(* CODESYS project CtaVisSymbols_2.0.0.0.library
   DocFormat: reStructuredText
   DefaultNamespace: CtaVisSymbols
   Version: 2.0.0.0
   Placeholder: CtaVisSymbols
   Company: CTA
   Description: Symbol Library der CTA
   CompiledLibraryCompatibilityVersion: CODESYS V3.5 SP16 Patch 3
   LanguageModelAttribute: qualified-access-only
   Title: CtaVisSymbols
   Author: SIS

Project tree, tasks and I/O mapping:
  libraries: CmpBitmapPool, 3.5.17.0 (System); VisuSymbols, 4.5.0.0 (System)
  40 Visualizations/
  30 Program Organization Units/
  00000000-0000-0000-0000-000000000000|D:\CoDeSys\LibrariesV3\trunk\Intern\CAA\CAA Template\3.4.0.0 draft\Placeholder.xml
  00000000-0000-0000-0000-000000000000|D:\CoDeSys\LibrariesV3\trunk\Intern\CAA\CAA Template\3.2.0.3 draft\Prefix.pdf
  00000000-0000-0000-0000-000000000000|D:\CoDeSys\LibrariesV3\trunk\Intern\CAA\CAA Template\3.5.2.0 draft\Placeholder.xml
  20 Structs/
  50 Images/
    image pool ImagePool
  10 Documenation/
    global variables VersionHistory
    global variables readMe
  21 Interface/
  11 Library Parameter/
  12 Konstanten/
  60 Textlisten/
  13 Globale Variablen/
  5ce3da45-db07-42e7-a21c-a00fff4ed8f6|Icons\Account.svg
  5ce3da45-db07-42e7-a21c-a00fff4ed8f6|Icons\alert.svg
  5ce3da45-db07-42e7-a21c-a00fff4ed8f6|Icons\alert_solo_black.svg
  5ce3da45-db07-42e7-a21c-a00fff4ed8f6|Icons\arrow-down.svg
  5ce3da45-db07-42e7-a21c-a00fff4ed8f6|Icons\arrow-down_solo_black.svg
  5ce3da45-db07-42e7-a21c-a00fff4ed8f6|Icons\arrow-down_square.svg
  5ce3da45-db07-42e7-a21c-a00fff4ed8f6|Icons\arrow-left.svg
  5ce3da45-db07-42e7-a21c-a00fff4ed8f6|Icons\arrow-left_solo_black.svg
  5ce3da45-db07-42e7-a21c-a00fff4ed8f6|Icons\arrow-left_square.svg
  5ce3da45-db07-42e7-a21c-a00fff4ed8f6|Icons\arrow-right_solo_black.svg
  5ce3da45-db07-42e7-a21c-a00fff4ed8f6|Icons\arrow-right_square.svg
  5ce3da45-db07-42e7-a21c-a00fff4ed8f6|Icons\arrow-up.svg
  5ce3da45-db07-42e7-a21c-a00fff4ed8f6|Icons\build.svg
  5ce3da45-db07-42e7-a21c-a00fff4ed8f6|Icons\calendar-range.svg
  5ce3da45-db07-42e7-a21c-a00fff4ed8f6|Icons\chart-bell-curve.svg
  5ce3da45-db07-42e7-a21c-a00fff4ed8f6|Icons\check.svg
  5ce3da45-db07-42e7-a21c-a00fff4ed8f6|Icons\check_solo_black.svg
  5ce3da45-db07-42e7-a21c-a00fff4ed8f6|Icons\clock-outline.svg
  5ce3da45-db07-42e7-a21c-a00fff4ed8f6|Icons\close.svg
  5ce3da45-db07-42e7-a21c-a00fff4ed8f6|Icons\close_solo_black.svg
  5ce3da45-db07-42e7-a21c-a00fff4ed8f6|Icons\CtaError.svg
  5ce3da45-db07-42e7-a21c-a00fff4ed8f6|Icons\CtaInfo.svg
  5ce3da45-db07-42e7-a21c-a00fff4ed8f6|Icons\CtaWarning.svg
  5ce3da45-db07-42e7-a21c-a00fff4ed8f6|Icons\database_black.svg
  5ce3da45-db07-42e7-a21c-a00fff4ed8f6|Icons\delete.svg
  5ce3da45-db07-42e7-a21c-a00fff4ed8f6|Icons\delete_solo_black.svg
  5ce3da45-db07-42e7-a21c-a00fff4ed8f6|Icons\dip-switch.svg
  5ce3da45-db07-42e7-a21c-a00fff4ed8f6|Icons\engine.svg
  5ce3da45-db07-42e7-a21c-a00fff4ed8f6|Icons\eye.svg
  5ce3da45-db07-42e7-a21c-a00fff4ed8f6|Icons\front_hand_Black.svg
  5ce3da45-db07-42e7-a21c-a00fff4ed8f6|Icons\front_hand_Yellow.svg
  5ce3da45-db07-42e7-a21c-a00fff4ed8f6|Icons\front_hand_Yellow_Off.svg
  5ce3da45-db07-42e7-a21c-a00fff4ed8f6|Icons\functions_black_24dp.svg
  5ce3da45-db07-42e7-a21c-a00fff4ed8f6|Icons\gear.svg
  5ce3da45-db07-42e7-a21c-a00fff4ed8f6|Icons\help.svg
  5ce3da45-db07-42e7-a21c-a00fff4ed8f6|Icons\home.svg
  5ce3da45-db07-42e7-a21c-a00fff4ed8f6|Icons\home_solo_black.svg
  5ce3da45-db07-42e7-a21c-a00fff4ed8f6|Icons\information-variant.svg
  5ce3da45-db07-42e7-a21c-a00fff4ed8f6|Icons\lan.svg
  5ce3da45-db07-42e7-a21c-a00fff4ed8f6|Icons\lightning-bolt-circle.svg
  5ce3da45-db07-42e7-a21c-a00fff4ed8f6|Icons\menu.svg
  5ce3da45-db07-42e7-a21c-a00fff4ed8f6|Icons\message.svg
  5ce3da45-db07-42e7-a21c-a00fff4ed8f6|Icons\message-alert-variant red.svg
  5ce3da45-db07-42e7-a21c-a00fff4ed8f6|Icons\message-alert-variant.svg
  5ce3da45-db07-42e7-a21c-a00fff4ed8f6|Icons\minus.svg
  5ce3da45-db07-42e7-a21c-a00fff4ed8f6|Icons\minus_solo_black.svg
  5ce3da45-db07-42e7-a21c-a00fff4ed8f6|Icons\plus.svg
  5ce3da45-db07-42e7-a21c-a00fff4ed8f6|Icons\plus_solo_black.svg
  5ce3da45-db07-42e7-a21c-a00fff4ed8f6|Icons\power.svg
  5ce3da45-db07-42e7-a21c-a00fff4ed8f6|Icons\power_solo_black.svg
  5ce3da45-db07-42e7-a21c-a00fff4ed8f6|Icons\refresh.svg
  5ce3da45-db07-42e7-a21c-a00fff4ed8f6|Icons\refresh_solo_black.svg
  5ce3da45-db07-42e7-a21c-a00fff4ed8f6|Icons\sd_card_black_24dp.svg
  5ce3da45-db07-42e7-a21c-a00fff4ed8f6|Icons\SearchFilter.svg
  5ce3da45-db07-42e7-a21c-a00fff4ed8f6|Icons\settings.svg
  5ce3da45-db07-42e7-a21c-a00fff4ed8f6|Icons\signal-celular-alt.svg
  5ce3da45-db07-42e7-a21c-a00fff4ed8f6|Icons\sine-wave.svg
  5ce3da45-db07-42e7-a21c-a00fff4ed8f6|Icons\toggle-switch.svg
  5ce3da45-db07-42e7-a21c-a00fff4ed8f6|Icons\toggle-switch-off.svg
  5ce3da45-db07-42e7-a21c-a00fff4ed8f6|Icons\Modbus_Organization_Logo.svg
  5ce3da45-db07-42e7-a21c-a00fff4ed8f6|Icons\CheckboxChecked_blue.svg
  5ce3da45-db07-42e7-a21c-a00fff4ed8f6|Icons\CheckboxUnchecked_withe.svg
  5ce3da45-db07-42e7-a21c-a00fff4ed8f6|Icons\lock_closed_black.svg
  5ce3da45-db07-42e7-a21c-a00fff4ed8f6|Icons\lock_open_black.svg
  5ce3da45-db07-42e7-a21c-a00fff4ed8f6|Icons\check_green.svg
  5ce3da45-db07-42e7-a21c-a00fff4ed8f6|Icons\close_red.svg
  5ce3da45-db07-42e7-a21c-a00fff4ed8f6|Icons\Sensor_Black.svg
  5ce3da45-db07-42e7-a21c-a00fff4ed8f6|Icons\filter_black.svg
  5ce3da45-db07-42e7-a21c-a00fff4ed8f6|Icons\notification_black.svg
  5ce3da45-db07-42e7-a21c-a00fff4ed8f6|Icons\CtaLogo.png
  5ce3da45-db07-42e7-a21c-a00fff4ed8f6|Icons\Edit_Stift.svg
  5ce3da45-db07-42e7-a21c-a00fff4ed8f6|Icons\Grafana_Logo.svg
  5ce3da45-db07-42e7-a21c-a00fff4ed8f6|Icons\InfluxDb_Logo.svg
  5ce3da45-db07-42e7-a21c-a00fff4ed8f6|Icons\hourglass_top.svg
  5ce3da45-db07-42e7-a21c-a00fff4ed8f6|Icons\Settings+.svg
  5ce3da45-db07-42e7-a21c-a00fff4ed8f6|Icons\Hourglass.gif
  5ce3da45-db07-42e7-a21c-a00fff4ed8f6|Icons\HandTapAwake.svg
  5ce3da45-db07-42e7-a21c-a00fff4ed8f6|Icons\gear_white.svg
  5ce3da45-db07-42e7-a21c-a00fff4ed8f6|S:\_Temporär_SIS\CtaCodesysLibrary\01_Library\CtaVisSymbols\Icons\SettingsSmall.svg
  5ce3da45-db07-42e7-a21c-a00fff4ed8f6|S:\_Temporär_SIS\CtaCodesysLibrary\01_Library\CtaVisSymbols\Icons\FileDescription.svg
  5ce3da45-db07-42e7-a21c-a00fff4ed8f6|S:\_Temporär_SIS\CtaCodesysLibrary\01_Library\CtaVisSymbols\Icons\Modbus_Organization_Logo_Short.svg
  5ce3da45-db07-42e7-a21c-a00fff4ed8f6|S:\_Temporär_SIS\CtaCodesysLibrary\01_Library\CtaVisSymbols\Icons\Chart.svg
  5ce3da45-db07-42e7-a21c-a00fff4ed8f6|\\cta.local\mue\Daten\200_Klima_Kälte\200_300_KK_CTA_Exklusiv_Elektro\01_Elektro\03_Software\00_CtaCodesysLibrary\01_Library\01 Source Code\CtaVisSymbols\Icons\ac_unit_40dp_ffffff_fill0_wght400_grad0_opsz40.svg
  5ce3da45-db07-42e7-a21c-a00fff4ed8f6|P:\200_Klima_Kälte\200_300_KK_CTA_Exklusiv_Elektro\01_Elektro\03_Software\00_CtaCodesysLibrary\01_Library\CtaVisSymbols\Icons\Account.svg
  5ce3da45-db07-42e7-a21c-a00fff4ed8f6|P:\200_Klima_Kälte\200_300_KK_CTA_Exklusiv_Elektro\01_Elektro\03_Software\00_CtaCodesysLibrary\01_Library\CtaVisSymbols\Icons\alert.svg
  5ce3da45-db07-42e7-a21c-a00fff4ed8f6|P:\200_Klima_Kälte\200_300_KK_CTA_Exklusiv_Elektro\01_Elektro\03_Software\00_CtaCodesysLibrary\01_Library\CtaVisSymbols\Icons\alert_solo_black.svg
  5ce3da45-db07-42e7-a21c-a00fff4ed8f6|P:\200_Klima_Kälte\200_300_KK_CTA_Exklusiv_Elektro\01_Elektro\03_Software\00_CtaCodesysLibrary\01_Library\CtaVisSymbols\Icons\arrow-down.svg
  5ce3da45-db07-42e7-a21c-a00fff4ed8f6|P:\200_Klima_Kälte\200_300_KK_CTA_Exklusiv_Elektro\01_Elektro\03_Software\00_CtaCodesysLibrary\01_Library\CtaVisSymbols\Icons\arrow-down_solo_black.svg
  5ce3da45-db07-42e7-a21c-a00fff4ed8f6|P:\200_Klima_Kälte\200_300_KK_CTA_Exklusiv_Elektro\01_Elektro\03_Software\00_CtaCodesysLibrary\01_Library\CtaVisSymbols\Icons\arrow-down_square.svg
  5ce3da45-db07-42e7-a21c-a00fff4ed8f6|P:\200_Klima_Kälte\200_300_KK_CTA_Exklusiv_Elektro\01_Elektro\03_Software\00_CtaCodesysLibrary\01_Library\CtaVisSymbols\Icons\arrow-left.svg
  5ce3da45-db07-42e7-a21c-a00fff4ed8f6|P:\200_Klima_Kälte\200_300_KK_CTA_Exklusiv_Elektro\01_Elektro\03_Software\00_CtaCodesysLibrary\01_Library\CtaVisSymbols\Icons\arrow-left_solo_black.svg
  5ce3da45-db07-42e7-a21c-a00fff4ed8f6|P:\200_Klima_Kälte\200_300_KK_CTA_Exklusiv_Elektro\01_Elektro\03_Software\00_CtaCodesysLibrary\01_Library\CtaVisSymbols\Icons\arrow-left_square.svg
  5ce3da45-db07-42e7-a21c-a00fff4ed8f6|P:\200_Klima_Kälte\200_300_KK_CTA_Exklusiv_Elektro\01_Elektro\03_Software\00_CtaCodesysLibrary\01_Library\CtaVisSymbols\Icons\arrow-right_solo_black.svg
  5ce3da45-db07-42e7-a21c-a00fff4ed8f6|P:\200_Klima_Kälte\200_300_KK_CTA_Exklusiv_Elektro\01_Elektro\03_Software\00_CtaCodesysLibrary\01_Library\CtaVisSymbols\Icons\arrow-right_square.svg
  5ce3da45-db07-42e7-a21c-a00fff4ed8f6|P:\200_Klima_Kälte\200_300_KK_CTA_Exklusiv_Elektro\01_Elektro\03_Software\00_CtaCodesysLibrary\01_Library\CtaVisSymbols\Icons\arrow-up.svg
  5ce3da45-db07-42e7-a21c-a00fff4ed8f6|P:\200_Klima_Kälte\200_300_KK_CTA_Exklusiv_Elektro\01_Elektro\03_Software\00_CtaCodesysLibrary\01_Library\CtaVisSymbols\Icons\build.svg
  5ce3da45-db07-42e7-a21c-a00fff4ed8f6|P:\200_Klima_Kälte\200_300_KK_CTA_Exklusiv_Elektro\01_Elektro\03_Software\00_CtaCodesysLibrary\01_Library\CtaVisSymbols\Icons\calendar-range.svg
  5ce3da45-db07-42e7-a21c-a00fff4ed8f6|P:\200_Klima_Kälte\200_300_KK_CTA_Exklusiv_Elektro\01_Elektro\03_Software\00_CtaCodesysLibrary\01_Library\CtaVisSymbols\Icons\Chart.svg
  5ce3da45-db07-42e7-a21c-a00fff4ed8f6|P:\200_Klima_Kälte\200_300_KK_CTA_Exklusiv_Elektro\01_Elektro\03_Software\00_CtaCodesysLibrary\01_Library\CtaVisSymbols\Icons\chart-bell-curve.svg
  5ce3da45-db07-42e7-a21c-a00fff4ed8f6|P:\200_Klima_Kälte\200_300_KK_CTA_Exklusiv_Elektro\01_Elektro\03_Software\00_CtaCodesysLibrary\01_Library\CtaVisSymbols\Icons\ChartLine.svg
  5ce3da45-db07-42e7-a21c-a00fff4ed8f6|P:\200_Klima_Kälte\200_300_KK_CTA_Exklusiv_Elektro\01_Elektro\03_Software\00_CtaCodesysLibrary\01_Library\CtaVisSymbols\Icons\chat_bubble_40dp_ffffff_fill0_wght400_grad0_opsz40.svg
  5ce3da45-db07-42e7-a21c-a00fff4ed8f6|P:\200_Klima_Kälte\200_300_KK_CTA_Exklusiv_Elektro\01_Elektro\03_Software\00_CtaCodesysLibrary\01_Library\CtaVisSymbols\Icons\check.svg
  5ce3da45-db07-42e7-a21c-a00fff4ed8f6|P:\200_Klima_Kälte\200_300_KK_CTA_Exklusiv_Elektro\01_Elektro\03_Software\00_CtaCodesysLibrary\01_Library\CtaVisSymbols\Icons\check_green.svg
  5ce3da45-db07-42e7-a21c-a00fff4ed8f6|P:\200_Klima_Kälte\200_300_KK_CTA_Exklusiv_Elektro\01_Elektro\03_Software\00_CtaCodesysLibrary\01_Library\CtaVisSymbols\Icons\check_solo_black.svg
  5ce3da45-db07-42e7-a21c-a00fff4ed8f6|P:\200_Klima_Kälte\200_300_KK_CTA_Exklusiv_Elektro\01_Elektro\03_Software\00_CtaCodesysLibrary\01_Library\CtaVisSymbols\Icons\checkboxchecked.svg
  5ce3da45-db07-42e7-a21c-a00fff4ed8f6|P:\200_Klima_Kälte\200_300_KK_CTA_Exklusiv_Elektro\01_Elektro\03_Software\00_CtaCodesysLibrary\01_Library\CtaVisSymbols\Icons\CheckboxChecked_blue.svg
  5ce3da45-db07-42e7-a21c-a00fff4ed8f6|P:\200_Klima_Kälte\200_300_KK_CTA_Exklusiv_Elektro\01_Elektro\03_Software\00_CtaCodesysLibrary\01_Library\CtaVisSymbols\Icons\checkboxchecked_def.svg
  5ce3da45-db07-42e7-a21c-a00fff4ed8f6|P:\200_Klima_Kälte\200_300_KK_CTA_Exklusiv_Elektro\01_Elektro\03_Software\00_CtaCodesysLibrary\01_Library\CtaVisSymbols\Icons\checkboxunchecked.svg
  5ce3da45-db07-42e7-a21c-a00fff4ed8f6|P:\200_Klima_Kälte\200_300_KK_CTA_Exklusiv_Elektro\01_Elektro\03_Software\00_CtaCodesysLibrary\01_Library\CtaVisSymbols\Icons\checkboxunchecked_def.svg
  5ce3da45-db07-42e7-a21c-a00fff4ed8f6|P:\200_Klima_Kälte\200_300_KK_CTA_Exklusiv_Elektro\01_Elektro\03_Software\00_CtaCodesysLibrary\01_Library\CtaVisSymbols\Icons\CheckboxUnchecked_withe.svg
  5ce3da45-db07-42e7-a21c-a00fff4ed8f6|P:\200_Klima_Kälte\200_300_KK_CTA_Exklusiv_Elektro\01_Elektro\03_Software\00_CtaCodesysLibrary\01_Library\CtaVisSymbols\Icons\clock-outline.svg
  5ce3da45-db07-42e7-a21c-a00fff4ed8f6|P:\200_Klima_Kälte\200_300_KK_CTA_Exklusiv_Elektro\01_Elektro\03_Software\00_CtaCodesysLibrary\01_Library\CtaVisSymbols\Icons\close.svg
  5ce3da45-db07-42e7-a21c-a00fff4ed8f6|P:\200_Klima_Kälte\200_300_KK_CTA_Exklusiv_Elektro\01_Elektro\03_Software\00_CtaCodesysLibrary\01_Library\CtaVisSymbols\Icons\close_red.svg
  5ce3da45-db07-42e7-a21c-a00fff4ed8f6|P:\200_Klima_Kälte\200_300_KK_CTA_Exklusiv_Elektro\01_Elektro\03_Software\00_CtaCodesysLibrary\01_Library\CtaVisSymbols\Icons\close_solo_black.svg
  5ce3da45-db07-42e7-a21c-a00fff4ed8f6|P:\200_Klima_Kälte\200_300_KK_CTA_Exklusiv_Elektro\01_Elektro\03_Software\00_CtaCodesysLibrary\01_Library\CtaVisSymbols\Icons\cloud_24dp_ffffff_fill0_wght400_grad0_opsz24.svg
  5ce3da45-db07-42e7-a21c-a00fff4ed8f6|P:\200_Klima_Kälte\200_300_KK_CTA_Exklusiv_Elektro\01_Elektro\03_Software\00_CtaCodesysLibrary\01_Library\CtaVisSymbols\Icons\cloudy_snowing_24dp_ffffff_fill0_wght400_grad0_opsz24.svg
  5ce3da45-db07-42e7-a21c-a00fff4ed8f6|P:\200_Klima_Kälte\200_300_KK_CTA_Exklusiv_Elektro\01_Elektro\03_Software\00_CtaCodesysLibrary\01_Library\CtaVisSymbols\Icons\CtaError.svg
  5ce3da45-db07-42e7-a21c-a00fff4ed8f6|P:\200_Klima_Kälte\200_300_KK_CTA_Exklusiv_Elektro\01_Elektro\03_Software\00_CtaCodesysLibrary\01_Library\CtaVisSymbols\Icons\CtaInfo.svg
  5ce3da45-db07-42e7-a21c-a00fff4ed8f6|P:\200_Klima_Kälte\200_300_KK_CTA_Exklusiv_Elektro\01_Elektro\03_Software\00_CtaCodesysLibrary\01_Library\CtaVisSymbols\Icons\CtaLogo.png
  5ce3da45-db07-42e7-a21c-a00fff4ed8f6|P:\200_Klima_Kälte\200_300_KK_CTA_Exklusiv_Elektro\01_Elektro\03_Software\00_CtaCodesysLibrary\01_Library\CtaVisSymbols\Icons\CtaWarning.svg
  5ce3da45-db07-42e7-a21c-a00fff4ed8f6|P:\200_Klima_Kälte\200_300_KK_CTA_Exklusiv_Elektro\01_Elektro\03_Software\00_CtaCodesysLibrary\01_Library\CtaVisSymbols\Icons\database_black.svg
  5ce3da45-db07-42e7-a21c-a00fff4ed8f6|P:\200_Klima_Kälte\200_300_KK_CTA_Exklusiv_Elektro\01_Elektro\03_Software\00_CtaCodesysLibrary\01_Library\CtaVisSymbols\Icons\delete.svg
  5ce3da45-db07-42e7-a21c-a00fff4ed8f6|P:\200_Klima_Kälte\200_300_KK_CTA_Exklusiv_Elektro\01_Elektro\03_Software\00_CtaCodesysLibrary\01_Library\CtaVisSymbols\Icons\delete_solo_black.svg
  5ce3da45-db07-42e7-a21c-a00fff4ed8f6|P:\200_Klima_Kälte\200_300_KK_CTA_Exklusiv_Elektro\01_Elektro\03_Software\00_CtaCodesysLibrary\01_Library\CtaVisSymbols\Icons\dictionary_40dp_ffffff_fill0_wght400_grad0_opsz40.svg
  5ce3da45-db07-42e7-a21c-a00fff4ed8f6|P:\200_Klima_Kälte\200_300_KK_CTA_Exklusiv_Elektro\01_Elektro\03_Software\00_CtaCodesysLibrary\01_Library\CtaVisSymbols\Icons\dip-switch.svg
  5ce3da45-db07-42e7-a21c-a00fff4ed8f6|P:\200_Klima_Kälte\200_300_KK_CTA_Exklusiv_Elektro\01_Elektro\03_Software\00_CtaCodesysLibrary\01_Library\CtaVisSymbols\Icons\Edit_Stift.svg
  5ce3da45-db07-42e7-a21c-a00fff4ed8f6|P:\200_Klima_Kälte\200_300_KK_CTA_Exklusiv_Elektro\01_Elektro\03_Software\00_CtaCodesysLibrary\01_Library\CtaVisSymbols\Icons\electric_bolt_24dp_000000_FILL0_wght400_GRAD0_opsz24.svg
  5ce3da45-db07-42e7-a21c-a00fff4ed8f6|P:\200_Klima_Kälte\200_300_KK_CTA_Exklusiv_Elektro\01_Elektro\03_Software\00_CtaCodesysLibrary\01_Library\CtaVisSymbols\Icons\engine.svg
  5ce3da45-db07-42e7-a21c-a00fff4ed8f6|P:\200_Klima_Kälte\200_300_KK_CTA_Exklusiv_Elektro\01_Elektro\03_Software\00_CtaCodesysLibrary\01_Library\CtaVisSymbols\Icons\engineering_40dp_ffffff_fill0_wght400_grad0_opsz40.svg
  5ce3da45-db07-42e7-a21c-a00fff4ed8f6|P:\200_Klima_Kälte\200_300_KK_CTA_Exklusiv_Elektro\01_Elektro\03_Software\00_CtaCodesysLibrary\01_Library\CtaVisSymbols\Icons\eye.svg
  5ce3da45-db07-42e7-a21c-a00fff4ed8f6|P:\200_Klima_Kälte\200_300_KK_CTA_Exklusiv_Elektro\01_Elektro\03_Software\00_CtaCodesysLibrary\01_Library\CtaVisSymbols\Icons\FileDescription.svg
  5ce3da45-db07-42e7-a21c-a00fff4ed8f6|P:\200_Klima_Kälte\200_300_KK_CTA_Exklusiv_Elektro\01_Elektro\03_Software\00_CtaCodesysLibrary\01_Library\CtaVisSymbols\Icons\filter_black.svg
  5ce3da45-db07-42e7-a21c-a00fff4ed8f6|P:\200_Klima_Kälte\200_300_KK_CTA_Exklusiv_Elektro\01_Elektro\03_Software\00_CtaCodesysLibrary\01_Library\CtaVisSymbols\Icons\foggy_24dp_ffffff_fill0_wght400_grad0_opsz24.svg
  5ce3da45-db07-42e7-a21c-a00fff4ed8f6|P:\200_Klima_Kälte\200_300_KK_CTA_Exklusiv_Elektro\01_Elektro\03_Software\00_CtaCodesysLibrary\01_Library\CtaVisSymbols\Icons\folder.svg
  5ce3da45-db07-42e7-a21c-a00fff4ed8f6|P:\200_Klima_Kälte\200_300_KK_CTA_Exklusiv_Elektro\01_Elektro\03_Software\00_CtaCodesysLibrary\01_Library\CtaVisSymbols\Icons\front_hand_Black.svg
  5ce3da45-db07-42e7-a21c-a00fff4ed8f6|P:\200_Klima_Kälte\200_300_KK_CTA_Exklusiv_Elektro\01_Elektro\03_Software\00_CtaCodesysLibrary\01_Library\CtaVisSymbols\Icons\front_hand_Yellow.svg
  5ce3da45-db07-42e7-a21c-a00fff4ed8f6|P:\200_Klima_Kälte\200_300_KK_CTA_Exklusiv_Elektro\01_Elektro\03_Software\00_CtaCodesysLibrary\01_Library\CtaVisSymbols\Icons\front_hand_Yellow_Off.svg
  5ce3da45-db07-42e7-a21c-a00fff4ed8f6|P:\200_Klima_Kälte\200_300_KK_CTA_Exklusiv_Elektro\01_Elektro\03_Software\00_CtaCodesysLibrary\01_Library\CtaVisSymbols\Icons\functions_black_24dp.svg
  5ce3da45-db07-42e7-a21c-a00fff4ed8f6|P:\200_Klima_Kälte\200_300_KK_CTA_Exklusiv_Elektro\01_Elektro\03_Software\00_CtaCodesysLibrary\01_Library\CtaVisSymbols\Icons\gear.svg
  5ce3da45-db07-42e7-a21c-a00fff4ed8f6|P:\200_Klima_Kälte\200_300_KK_CTA_Exklusiv_Elektro\01_Elektro\03_Software\00_CtaCodesysLibrary\01_Library\CtaVisSymbols\Icons\gear_white.svg
  5ce3da45-db07-42e7-a21c-a00fff4ed8f6|P:\200_Klima_Kälte\200_300_KK_CTA_Exklusiv_Elektro\01_Elektro\03_Software\00_CtaCodesysLibrary\01_Library\CtaVisSymbols\Icons\Grafana_Logo.svg
  5ce3da45-db07-42e7-a21c-a00fff4ed8f6|P:\200_Klima_Kälte\200_300_KK_CTA_Exklusiv_Elektro\01_Elektro\03_Software\00_CtaCodesysLibrary\01_Library\CtaVisSymbols\Icons\HandTapAwake.svg
  5ce3da45-db07-42e7-a21c-a00fff4ed8f6|P:\200_Klima_Kälte\200_300_KK_CTA_Exklusiv_Elektro\01_Elektro\03_Software\00_CtaCodesysLibrary\01_Library\CtaVisSymbols\Icons\help.svg
  5ce3da45-db07-42e7-a21c-a00fff4ed8f6|P:\200_Klima_Kälte\200_300_KK_CTA_Exklusiv_Elektro\01_Elektro\03_Software\00_CtaCodesysLibrary\01_Library\CtaVisSymbols\Icons\home.svg
  5ce3da45-db07-42e7-a21c-a00fff4ed8f6|P:\200_Klima_Kälte\200_300_KK_CTA_Exklusiv_Elektro\01_Elektro\03_Software\00_CtaCodesysLibrary\01_Library\CtaVisSymbols\Icons\home_40dp_ffffff_fill0_wght400_grad0_opsz40.svg
  5ce3da45-db07-42e7-a21c-a00fff4ed8f6|P:\200_Klima_Kälte\200_300_KK_CTA_Exklusiv_Elektro\01_Elektro\03_Software\00_CtaCodesysLibrary\01_Library\CtaVisSymbols\Icons\home_solo_black.svg
  5ce3da45-db07-42e7-a21c-a00fff4ed8f6|P:\200_Klima_Kälte\200_300_KK_CTA_Exklusiv_Elektro\01_Elektro\03_Software\00_CtaCodesysLibrary\01_Library\CtaVisSymbols\Icons\Hourglass.gif
  5ce3da45-db07-42e7-a21c-a00fff4ed8f6|P:\200_Klima_Kälte\200_300_KK_CTA_Exklusiv_Elektro\01_Elektro\03_Software\00_CtaCodesysLibrary\01_Library\CtaVisSymbols\Icons\hourglass_top.svg
  5ce3da45-db07-42e7-a21c-a00fff4ed8f6|P:\200_Klima_Kälte\200_300_KK_CTA_Exklusiv_Elektro\01_Elektro\03_Software\00_CtaCodesysLibrary\01_Library\CtaVisSymbols\Icons\hub_20dp_ffffff_fill0_wght400_grad0_opsz20.svg
  5ce3da45-db07-42e7-a21c-a00fff4ed8f6|P:\200_Klima_Kälte\200_300_KK_CTA_Exklusiv_Elektro\01_Elektro\03_Software\00_CtaCodesysLibrary\01_Library\CtaVisSymbols\Icons\InfluxDb_Logo.svg
  5ce3da45-db07-42e7-a21c-a00fff4ed8f6|P:\200_Klima_Kälte\200_300_KK_CTA_Exklusiv_Elektro\01_Elektro\03_Software\00_CtaCodesysLibrary\01_Library\CtaVisSymbols\Icons\information-variant.svg
  5ce3da45-db07-42e7-a21c-a00fff4ed8f6|P:\200_Klima_Kälte\200_300_KK_CTA_Exklusiv_Elektro\01_Elektro\03_Software\00_CtaCodesysLibrary\01_Library\CtaVisSymbols\Icons\instant_mix_40dp_ffffff_fill0_wght400_grad0_opsz40.svg
  5ce3da45-db07-42e7-a21c-a00fff4ed8f6|P:\200_Klima_Kälte\200_300_KK_CTA_Exklusiv_Elektro\01_Elektro\03_Software\00_CtaCodesysLibrary\01_Library\CtaVisSymbols\Icons\lan.svg
  5ce3da45-db07-42e7-a21c-a00fff4ed8f6|P:\200_Klima_Kälte\200_300_KK_CTA_Exklusiv_Elektro\01_Elektro\03_Software\00_CtaCodesysLibrary\01_Library\CtaVisSymbols\Icons\lan_40dp_ffffff_fill0_wght400_grad0_opsz40.svg
  5ce3da45-db07-42e7-a21c-a00fff4ed8f6|P:\200_Klima_Kälte\200_300_KK_CTA_Exklusiv_Elektro\01_Elektro\03_Software\00_CtaCodesysLibrary\01_Library\CtaVisSymbols\Icons\language_50dp_ffffff_fill0_wght400_grad0_opsz48.svg
  5ce3da45-db07-42e7-a21c-a00fff4ed8f6|P:\200_Klima_Kälte\200_300_KK_CTA_Exklusiv_Elektro\01_Elektro\03_Software\00_CtaCodesysLibrary\01_Library\CtaVisSymbols\Icons\lightning-bolt-circle.svg
  5ce3da45-db07-42e7-a21c-a00fff4ed8f6|P:\200_Klima_Kälte\200_300_KK_CTA_Exklusiv_Elektro\01_Elektro\03_Software\00_CtaCodesysLibrary\01_Library\CtaVisSymbols\Icons\link_24dp_5f6368_fill0_wght400_grad0_opsz24.svg
  5ce3da45-db07-42e7-a21c-a00fff4ed8f6|P:\200_Klima_Kälte\200_300_KK_CTA_Exklusiv_Elektro\01_Elektro\03_Software\00_CtaCodesysLibrary\01_Library\CtaVisSymbols\Icons\link_off_24dp_5f6368_fill0_wght400_grad0_opsz24.svg
  5ce3da45-db07-42e7-a21c-a00fff4ed8f6|P:\200_Klima_Kälte\200_300_KK_CTA_Exklusiv_Elektro\01_Elektro\03_Software\00_CtaCodesysLibrary\01_Library\CtaVisSymbols\Icons\lock_closed_black.svg
  5ce3da45-db07-42e7-a21c-a00fff4ed8f6|P:\200_Klima_Kälte\200_300_KK_CTA_Exklusiv_Elektro\01_Elektro\03_Software\00_CtaCodesysLibrary\01_Library\CtaVisSymbols\Icons\lock_open_black.svg
  5ce3da45-db07-42e7-a21c-a00fff4ed8f6|P:\200_Klima_Kälte\200_300_KK_CTA_Exklusiv_Elektro\01_Elektro\03_Software\00_CtaCodesysLibrary\01_Library\CtaVisSymbols\Icons\lockicon.svg
  5ce3da45-db07-42e7-a21c-a00fff4ed8f6|P:\200_Klima_Kälte\200_300_KK_CTA_Exklusiv_Elektro\01_Elektro\03_Software\00_CtaCodesysLibrary\01_Library\CtaVisSymbols\Icons\logout_50dp_ffffff_fill0_wght400_grad0_opsz48.svg
  5ce3da45-db07-42e7-a21c-a00fff4ed8f6|P:\200_Klima_Kälte\200_300_KK_CTA_Exklusiv_Elektro\01_Elektro\03_Software\00_CtaCodesysLibrary\01_Library\CtaVisSymbols\Icons\memory_20dp_ffffff_fill0_wght400_grad0_opsz20.svg
  5ce3da45-db07-42e7-a21c-a00fff4ed8f6|P:\200_Klima_Kälte\200_300_KK_CTA_Exklusiv_Elektro\01_Elektro\03_Software\00_CtaCodesysLibrary\01_Library\CtaVisSymbols\Icons\menu.svg
  5ce3da45-db07-42e7-a21c-a00fff4ed8f6|P:\200_Klima_Kälte\200_300_KK_CTA_Exklusiv_Elektro\01_Elektro\03_Software\00_CtaCodesysLibrary\01_Library\CtaVisSymbols\Icons\menu_50dp_ffffff_fill0_wght400_grad0_opsz48.svg
  5ce3da45-db07-42e7-a21c-a00fff4ed8f6|P:\200_Klima_Kälte\200_300_KK_CTA_Exklusiv_Elektro\01_Elektro\03_Software\00_CtaCodesysLibrary\01_Library\CtaVisSymbols\Icons\menu_open_50dp_ffffff_fill0_wght400_grad0_opsz48.svg
  5ce3da45-db07-42e7-a21c-a00fff4ed8f6|P:\200_Klima_Kälte\200_300_KK_CTA_Exklusiv_Elektro\01_Elektro\03_Software\00_CtaCodesysLibrary\01_Library\CtaVisSymbols\Icons\message.svg
  5ce3da45-db07-42e7-a21c-a00fff4ed8f6|P:\200_Klima_Kälte\200_300_KK_CTA_Exklusiv_Elektro\01_Elektro\03_Software\00_CtaCodesysLibrary\01_Library\CtaVisSymbols\Icons\message-alert-variant red.svg
  5ce3da45-db07-42e7-a21c-a00fff4ed8f6|P:\200_Klima_Kälte\200_300_KK_CTA_Exklusiv_Elektro\01_Elektro\03_Software\00_CtaCodesysLibrary\01_Library\CtaVisSymbols\Icons\message-alert-variant.svg
  5ce3da45-db07-42e7-a21c-a00fff4ed8f6|P:\200_Klima_Kälte\200_300_KK_CTA_Exklusiv_Elektro\01_Elektro\03_Software\00_CtaCodesysLibrary\01_Library\CtaVisSymbols\Icons\minus.svg
  5ce3da45-db07-42e7-a21c-a00fff4ed8f6|P:\200_Klima_Kälte\200_300_KK_CTA_Exklusiv_Elektro\01_Elektro\03_Software\00_CtaCodesysLibrary\01_Library\CtaVisSymbols\Icons\minus_solo_black.svg
  5ce3da45-db07-42e7-a21c-a00fff4ed8f6|P:\200_Klima_Kälte\200_300_KK_CTA_Exklusiv_Elektro\01_Elektro\03_Software\00_CtaCodesysLibrary\01_Library\CtaVisSymbols\Icons\Modbus_Organization_Logo.svg
  5ce3da45-db07-42e7-a21c-a00fff4ed8f6|P:\200_Klima_Kälte\200_300_KK_CTA_Exklusiv_Elektro\01_Elektro\03_Software\00_CtaCodesysLibrary\01_Library\CtaVisSymbols\Icons\Modbus_Organization_Logo_Short.svg
  5ce3da45-db07-42e7-a21c-a00fff4ed8f6|P:\200_Klima_Kälte\200_300_KK_CTA_Exklusiv_Elektro\01_Elektro\03_Software\00_CtaCodesysLibrary\01_Library\CtaVisSymbols\Icons\mode_cool_24dp_ffffff_fill0_wght400_grad0_opsz24.svg
  5ce3da45-db07-42e7-a21c-a00fff4ed8f6|P:\200_Klima_Kälte\200_300_KK_CTA_Exklusiv_Elektro\01_Elektro\03_Software\00_CtaCodesysLibrary\01_Library\CtaVisSymbols\Icons\monitoring_40dp_ffffff_fill0_wght400_grad0_opsz40.svg
  5ce3da45-db07-42e7-a21c-a00fff4ed8f6|P:\200_Klima_Kälte\200_300_KK_CTA_Exklusiv_Elektro\01_Elektro\03_Software\00_CtaCodesysLibrary\01_Library\CtaVisSymbols\Icons\notification_black.svg
  5ce3da45-db07-42e7-a21c-a00fff4ed8f6|P:\200_Klima_Kälte\200_300_KK_CTA_Exklusiv_Elektro\01_Elektro\03_Software\00_CtaCodesysLibrary\01_Library\CtaVisSymbols\Icons\partly_cloudy_day_24dp_ffffff_fill0_wght400_grad0_opsz24.svg
  5ce3da45-db07-42e7-a21c-a00fff4ed8f6|P:\200_Klima_Kälte\200_300_KK_CTA_Exklusiv_Elektro\01_Elektro\03_Software\00_CtaCodesysLibrary\01_Library\CtaVisSymbols\Icons\person_50dp_ffffff_fill0_wght400_grad0_opsz48.svg
  5ce3da45-db07-42e7-a21c-a00fff4ed8f6|P:\200_Klima_Kälte\200_300_KK_CTA_Exklusiv_Elektro\01_Elektro\03_Software\00_CtaCodesysLibrary\01_Library\CtaVisSymbols\Icons\plus.svg
  5ce3da45-db07-42e7-a21c-a00fff4ed8f6|P:\200_Klima_Kälte\200_300_KK_CTA_Exklusiv_Elektro\01_Elektro\03_Software\00_CtaCodesysLibrary\01_Library\CtaVisSymbols\Icons\plus_solo_black.svg
  5ce3da45-db07-42e7-a21c-a00fff4ed8f6|P:\200_Klima_Kälte\200_300_KK_CTA_Exklusiv_Elektro\01_Elektro\03_Software\00_CtaCodesysLibrary\01_Library\CtaVisSymbols\Icons\power.svg
  5ce3da45-db07-42e7-a21c-a00fff4ed8f6|P:\200_Klima_Kälte\200_300_KK_CTA_Exklusiv_Elektro\01_Elektro\03_Software\00_CtaCodesysLibrary\01_Library\CtaVisSymbols\Icons\power_solo_black.svg
  5ce3da45-db07-42e7-a21c-a00fff4ed8f6|P:\200_Klima_Kälte\200_300_KK_CTA_Exklusiv_Elektro\01_Elektro\03_Software\00_CtaCodesysLibrary\01_Library\CtaVisSymbols\Icons\radiobuttonchecked.svg
  5ce3da45-db07-42e7-a21c-a00fff4ed8f6|P:\200_Klima_Kälte\200_300_KK_CTA_Exklusiv_Elektro\01_Elektro\03_Software\00_CtaCodesysLibrary\01_Library\CtaVisSymbols\Icons\radiobuttonunchecked.svg
  5ce3da45-db07-42e7-a21c-a00fff4ed8f6|P:\200_Klima_Kälte\200_300_KK_CTA_Exklusiv_Elektro\01_Elektro\03_Software\00_CtaCodesysLibrary\01_Library\CtaVisSymbols\Icons\rainy_24dp_ffffff_fill0_wght400_grad0_opsz24.svg
  5ce3da45-db07-42e7-a21c-a00fff4ed8f6|P:\200_Klima_Kälte\200_300_KK_CTA_Exklusiv_Elektro\01_Elektro\03_Software\00_CtaCodesysLibrary\01_Library\CtaVisSymbols\Icons\refresh.svg
  5ce3da45-db07-42e7-a21c-a00fff4ed8f6|P:\200_Klima_Kälte\200_300_KK_CTA_Exklusiv_Elektro\01_Elektro\03_Software\00_CtaCodesysLibrary\01_Library\CtaVisSymbols\Icons\refresh_solo_black.svg
  5ce3da45-db07-42e7-a21c-a00fff4ed8f6|P:\200_Klima_Kälte\200_300_KK_CTA_Exklusiv_Elektro\01_Elektro\03_Software\00_CtaCodesysLibrary\01_Library\CtaVisSymbols\Icons\sd_card_black_24dp.svg
  5ce3da45-db07-42e7-a21c-a00fff4ed8f6|P:\200_Klima_Kälte\200_300_KK_CTA_Exklusiv_Elektro\01_Elektro\03_Software\00_CtaCodesysLibrary\01_Library\CtaVisSymbols\Icons\SearchFilter.svg
  5ce3da45-db07-42e7-a21c-a00fff4ed8f6|P:\200_Klima_Kälte\200_300_KK_CTA_Exklusiv_Elektro\01_Elektro\03_Software\00_CtaCodesysLibrary\01_Library\CtaVisSymbols\Icons\Sensor_Black.svg
  5ce3da45-db07-42e7-a21c-a00fff4ed8f6|P:\200_Klima_Kälte\200_300_KK_CTA_Exklusiv_Elektro\01_Elektro\03_Software\00_CtaCodesysLibrary\01_Library\CtaVisSymbols\Icons\settings.svg
  5ce3da45-db07-42e7-a21c-a00fff4ed8f6|P:\200_Klima_Kälte\200_300_KK_CTA_Exklusiv_Elektro\01_Elektro\03_Software\00_CtaCodesysLibrary\01_Library\CtaVisSymbols\Icons\settings_40dp_ffffff_fill0_wght400_grad0_opsz40.svg
  5ce3da45-db07-42e7-a21c-a00fff4ed8f6|P:\200_Klima_Kälte\200_300_KK_CTA_Exklusiv_Elektro\01_Elektro\03_Software\00_CtaCodesysLibrary\01_Library\CtaVisSymbols\Icons\settings_power_40dp_ffffff_fill0_wght400_grad0_opsz40.svg
  5ce3da45-db07-42e7-a21c-a00fff4ed8f6|P:\200_Klima_Kälte\200_300_KK_CTA_Exklusiv_Elektro\01_Elektro\03_Software\00_CtaCodesysLibrary\01_Library\CtaVisSymbols\Icons\Settings+.svg
  5ce3da45-db07-42e7-a21c-a00fff4ed8f6|P:\200_Klima_Kälte\200_300_KK_CTA_Exklusiv_Elektro\01_Elektro\03_Software\00_CtaCodesysLibrary\01_Library\CtaVisSymbols\Icons\SettingsSmall.svg
  5ce3da45-db07-42e7-a21c-a00fff4ed8f6|P:\200_Klima_Kälte\200_300_KK_CTA_Exklusiv_Elektro\01_Elektro\03_Software\00_CtaCodesysLibrary\01_Library\CtaVisSymbols\Icons\signal-celular-alt.svg
  5ce3da45-db07-42e7-a21c-a00fff4ed8f6|P:\200_Klima_Kälte\200_300_KK_CTA_Exklusiv_Elektro\01_Elektro\03_Software\00_CtaCodesysLibrary\01_Library\CtaVisSymbols\Icons\sine-wave.svg
  5ce3da45-db07-42e7-a21c-a00fff4ed8f6|P:\200_Klima_Kälte\200_300_KK_CTA_Exklusiv_Elektro\01_Elektro\03_Software\00_CtaCodesysLibrary\01_Library\CtaVisSymbols\Icons\sunny_24dp_ffffff_fill0_wght400_grad0_opsz24.svg
  5ce3da45-db07-42e7-a21c-a00fff4ed8f6|P:\200_Klima_Kälte\200_300_KK_CTA_Exklusiv_Elektro\01_Elektro\03_Software\00_CtaCodesysLibrary\01_Library\CtaVisSymbols\Icons\thunderstorm_24dp_ffffff_fill0_wght400_grad0_opsz24.svg
  5ce3da45-db07-42e7-a21c-a00fff4ed8f6|P:\200_Klima_Kälte\200_300_KK_CTA_Exklusiv_Elektro\01_Elektro\03_Software\00_CtaCodesysLibrary\01_Library\CtaVisSymbols\Icons\toggle-switch.svg
  5ce3da45-db07-42e7-a21c-a00fff4ed8f6|P:\200_Klima_Kälte\200_300_KK_CTA_Exklusiv_Elektro\01_Elektro\03_Software\00_CtaCodesysLibrary\01_Library\CtaVisSymbols\Icons\toggle-switch-off.svg
  5ce3da45-db07-42e7-a21c-a00fff4ed8f6|P:\200_Klima_Kälte\200_300_KK_CTA_Exklusiv_Elektro\01_Elektro\03_Software\00_CtaCodesysLibrary\01_Library\CtaVisSymbols\Icons\usericon.svg
  5ce3da45-db07-42e7-a21c-a00fff4ed8f6|P:\200_Klima_Kälte\200_300_KK_CTA_Exklusiv_Elektro\01_Elektro\03_Software\00_CtaCodesysLibrary\01_Library\CtaVisSymbols\Icons\water_pump_40dp_ffffff_fill0_wght400_grad0_opsz40.svg
  5ce3da45-db07-42e7-a21c-a00fff4ed8f6|P:\200_Klima_Kälte\200_300_KK_CTA_Exklusiv_Elektro\01_Elektro\03_Software\00_CtaCodesysLibrary\01_Library\CtaVisSymbols\Icons\valve_24dp_000000_FILL0_wght400_GRAD0_opsz24.svg
  5ce3da45-db07-42e7-a21c-a00fff4ed8f6|\\cta.local\mue\Daten\200_Klima_Kälte\200_300_KK_CTA_Exklusiv_Elektro\01_Elektro\03_Software\00_CtaCodesysLibrary\01_Library\01 Source Code\CtaVisSymbols\Icons\deployed_code_update_40dp_FFFFFF_FILL0_wght400_GRAD0_opsz40.svg
  5ce3da45-db07-42e7-a21c-a00fff4ed8f6|\\cta.local\mue\Daten\200_Klima_Kälte\200_300_KK_CTA_Exklusiv_Elektro\01_Elektro\03_Software\00_CtaCodesysLibrary\01_Library\01 Source Code\CtaVisSymbols\Icons\admin_panel_settings_40dp_ffffff_fill0_wght400_grad0_opsz40.svg
*)

// 10 Documenation/VersionHistory
(* 

.. image:: ../../Images/CTA_Logo.jpg
   :align: right
   :width: 15% 

**Vorlage**   


============ =========== =========== ============================================
**Date**     **Version** **Author**  **Change**
------------ ----------- ----------- --------------------------------------------
04.03.2021   0.0.0.0     SIS         Vorlage erstellt

============ =========== =========== ============================================


*)
VAR_GLOBAL
    stInfo : STRING:= '0.0.0.0, Vorlage, CTA';
END_VAR

// 10 Documenation/readMe
(*

**ReadMe**
 
|	**Empfehlung**
|
|	Dokumentrieren Sie die Library für eine nachhaltige Entwicklung
|     
| *Beispiel*
| 
| Dies ist die Vorlage Library der CTA. Erstellen Sie ihre Library anhand dieser Vorlage.
*)

VAR_GLOBAL
    xReadMeDone              :   BOOL;
END_VAR
